{attribute 'qualified_only'}
VAR_GLOBAL
//Vision_Bool
	HaertBeat								:	BOOL	;
	HaertBeat_ON							:	BOOL	;
	HaertBeat_OFF							:	BOOL	;
	Data_Read_Comp							:	BOOL	;
	Data_Read_OK							:	BOOL	;
	Data_Read_NG							:	BOOL	;
	Axis02_Data_Apply_Comp					:	BOOL	;
	Axis03_Data_Apply_Comp					:	BOOL	;
	Axis05_Data_Apply_Comp					:	BOOL	;
	Cam_Trigger					AT%Q*		:	BOOL	;
	Get_Frame								:	BOOL	;
	Vision_OK								:	BOOL	;
	Vision_NG								:	BOOL	;
	Run										:	BOOL	;
	Vision_Light_ON				AT%Q*		:	BOOL 	;
	Data_Copy_Comp							:	BOOL	;
	Data_Empty								:	BOOL	;
	
//Vision Data
	Data_Read_X								:	LREAL	;
	Data_Read_Y								:	LREAL	;
	Data_Read_R								:	LREAL	;
	Press_Speed								:	LREAL	;
	Travel_Distance							:	LREAL	;
	Target_Distance							:	LREAL	;
	Target_X_Real_Position_Data				:	LREAL	;
	Moving_Time								:	LREAL	;
	FrameCount								:	LREAL	;
	TotalSpeed								:	LREAL	;
	Average_Speed							:	LREAL	;
	Get_Frame_Time							:	LREAL	;
	ON_Delay_Time							:	LREAL	;
	Start_Pos_Data							:	LREAL	;
	Encoder_DATA03							:	LREAL	;

//Vision_Status
	Vision_Alarm_Code						:	INT		;
	Axis02_Calibration_Position_Data		:	LREAL	;
	Axis03_Calibration_Position_Data		:	LREAL	;
	Axis05_Calibration_Position_Data		:	LREAL	;
	Axis02_Calibration_Position_Data_Old	:	LREAL	;
	Axis03_Calibration_Position_Data_Old	:	LREAL	;
	Axis05_Calibration_Position_Data_Old	:	LREAL	;
	Axis02_Tool_Change_Position_Data		:	LREAL	;
	Axis03_Tool_Change_Position_Data		:	LREAL	;
	Axis04_Tool_Change_Position_Data		:	LREAL	;
	
	
//Vision_Data_Buffer

	Data_Buffer_X							:	LREAL	;
	Data_Buffer_Y							:	LREAL	;
	Data_Buffer_R							:	LREAL	;
	
	
	Encoder_DATA01							: ARRAY[1..5] OF LREAL;
	Encoder_DATA02							:	LREAL	;
	
	Cam_Trigger_Length						:	LREAL	;


	Data_Check: BOOL;
	Vision_Start_Sensor: BOOL;
END_VAR
VAR_GLOBAL PERSISTENT
	DATA_COUNT								: 	INT;

	
END_VAR

(* stored: Version 1.1.0.1, ProductVersion 3.1.4024.15
   GVL GVL_Vision: Id {aacb4183-bf71-4ea7-aa39-f263d21233e2} *)
